INTERFACE I_ExternalLogger

METHOD AddToLog
VAR_IN_OUT
   Message : T_MaxString;
END_VAR
VAR_INPUT
   LogSeverity : E_LogSeverity;
END_VAR
END_METHOD

END_INTERFACE

(* stored: Version 1.1.0.1, ProductVersion 3.1.4026.12
   Itf I_ExternalLogger: Id {d75d9843-761c-0d34-140b-aa07a979d486}
   Method AddToLog: Id {757471e8-b729-0d32-3eb4-5b32f786d76d} *)
